{attribute addProperty BoxType "EL2202-0000-0016"}
{attribute addProperty Id "ChannelAT %Q*ARRAY[0..2] OF Channel_D43BF62A3240WcStateAT %I*WcState_28A8677510.1250InfoDataAT %I*InfoData_192954DE1620"}
{attribute addProperty CRC "372252385"}
{attribute addProperty SizeInBites "49"}
{attribute addProperty SizeInBytes "6.125"}
TYPE EL2202_B7733B6A :
STRUCT
	{attribute addProperty Name "Channel"}
	Channel : ARRAY[0..2] OF Channel_D43BF62A;
	{attribute addProperty Name "WcState"}
	WcState : WcState_28A86775;
	{attribute addProperty Name "InfoData"}
	InfoData : InfoData_192954DE;
END_STRUCT
END_TYPE

(* stored: Version 1.2.0.0, ProductVersion 3.1.4024.9
   DUT EL2202_B7733B6A: Id {8d81ad63-5f84-4126-9e0a-3176a8a35357} *)
